INTERFACE I_Mover EXTENDS I_Base

{attribute 'monitoring':='call'}
PROPERTY Parameters : I_ParameterPosition
GET
END_GET
SET
END_SET
END_PROPERTY

{attribute 'monitoring':='call'}
PROPERTY Status : I_ParameterPositionGetter
GET
END_GET
END_PROPERTY

END_INTERFACE

(* stored: Version 1.1.0.1
   Itf I_Mover: Id {9bb10a3f-2f99-4fcb-8194-d43da0221a55}
   Property Parameters: Id {16171c9e-fc79-404d-a79c-639c3690963c}
   Get Get: Id {a3e7bdb5-610a-4ec0-bd86-7e73a80f3402}
   Set Set: Id {da3fe086-677b-4248-a266-7327bf7e9e4f}
   Property Status: Id {40b7d67b-24e5-44f2-a819-c4aa335e8856}
   Get Get: Id {e00bb714-94a6-40e5-9449-9c78977bad5f} *)
